(* IEC 61131-3 sources: SmartHomeNew/snapshots/2026-04-22, 17 files *)

(* ---- E_TwoFactor_Method.dut ---- *)
{attribute 'strict'}
TYPE E_TwoFactor_Method :
(
    TF_METHOD_NONE := 0,
    TF_METHOD_RFID := 1,
    TF_METHOD_TOTP := 2,
    TF_METHOD_BOTH := 3
) USINT;
END_TYPE

(* ---- ST_Heating_Config.dut ---- *)
{attribute 'pack_mode' := '1'}
TYPE ST_Heating_Config :
STRUCT
    Weather_Comp_Enabled : BOOL := TRUE;
    Weather_Coef : REAL := 0.1;
    Freeze_Threshold : REAL := 7.0;
    Overheat_Threshold : REAL := 45.0;
    Night_Reduction : REAL := 3.0;
    Target_Floor_Temp : REAL := 28.0;
    Target_Room_Temp : REAL := 22.0;
    Hysteresis : REAL := 0.5;
END_STRUCT
END_TYPE

(* ---- ST_System_State_Snapshot.dut ---- *)
{attribute 'pack_mode' := '1'}
TYPE ST_System_State_Snapshot :
STRUCT
    System_Time_MS : UDINT;
    Current_Scenario : E_SCENARIO_TYPE;
    Security_Armed : BOOL;
    Active_Alarms : INT;
    // Критические состояния для синхронизации
    Zone_Valves : ARRAY[1..8] OF BOOL;
    Manifold_Pumps : ARRAY[1..GVL_CONSTANTS.C_MAX_MANIFOLDS] OF BOOL;
    Lighting_States : ARRAY[1..32] OF BYTE;
    Blinds_Positions : ARRAY[1..GVL_CONSTANTS.C_MAX_BLINDS] OF BYTE;
    Socket_States : ARRAY[1..GVL_CONSTANTS.C_MAX_SOCKETS] OF BOOL;
    Gas_Valve_Closed : BOOL;
    Water_Valves_Closed : BOOL;
    Version : UDINT; // Версия состояния для разрешения конфликтов
END_STRUCT
END_TYPE

(* ---- ST_Zone_Sensors.dut ---- *)
{attribute 'pack_mode' := '1'}
TYPE ST_Zone_Sensors :
STRUCT
    Temp_Room : REAL;
    Temp_Floor : REAL;
    Motion_Active : BOOL;
    Switch_Physical : BOOL;
    Light_State : BOOL;
    Maintenance : ST_Component_Maintenance;
END_STRUCT
END_TYPE

(* ---- FB_Fault_Logger.st ---- *)
FUNCTION_BLOCK FB_Fault_Logger
VAR_INPUT
    VI_Severity  : E_System_Severity;
    VI_RootCause : E_System_Root_Cause;
    VI_Time_MS   : UDINT;
END_VAR

VAR_OUTPUT
    VO_Last_Event_Text : STRING(200);
    VO_Event_Count     : UINT;
    VO_Last_Index      : UINT;

    VO_Event_Time_MS   : ARRAY[1..16] OF UDINT;
    VO_Event_Severity  : ARRAY[1..16] OF E_System_Severity;
    VO_Event_RootCause : ARRAY[1..16] OF E_System_Root_Cause;
    VO_Event_Text      : ARRAY[1..16] OF STRING(200);
END_VAR

VAR
    L_Last_Severity  : E_System_Severity;
    L_Last_RootCause : E_System_Root_Cause;
    L_Write_Index    : UINT := 0;
    L_Event_Text     : STRING(200);
END_VAR

L_Event_Text := '';

IF (VI_Severity <> L_Last_Severity) OR (VI_RootCause <> L_Last_RootCause) THEN
    CASE VI_RootCause OF
        E_System_Root_Cause.ROOT_FIRE:
            L_Event_Text := 'EVENT: FIRE DETECTED';
        E_System_Root_Cause.ROOT_GAS_LEAK:
            L_Event_Text := 'EVENT: GAS LEAK';
        E_System_Root_Cause.ROOT_CO_CRITICAL:
            L_Event_Text := 'EVENT: CO CRITICAL';
        E_System_Root_Cause.ROOT_CO_WARNING:
            L_Event_Text := 'EVENT: CO WARNING';
        E_System_Root_Cause.ROOT_WATER_LEAK:
            L_Event_Text := 'EVENT: WATER LEAK';
        E_System_Root_Cause.ROOT_SENSOR_FAULT:
            L_Event_Text := 'EVENT: SENSOR FAULT';
        E_System_Root_Cause.ROOT_IO_OFFLINE:
            L_Event_Text := 'EVENT: IO OFFLINE';
        E_System_Root_Cause.ROOT_COMM_FAULT:
            L_Event_Text := 'EVENT: COMM FAULT';
        E_System_Root_Cause.ROOT_WATCHDOG_FAULT:
            L_Event_Text := 'EVENT: WATCHDOG FAULT';
        E_System_Root_Cause.ROOT_SUBSYSTEM_FAULT:
            L_Event_Text := 'EVENT: SUBSYSTEM FAULT';
        ELSE
            L_Event_Text := 'EVENT: SYSTEM STATE CHANGE';
    END_CASE;

    L_Write_Index := L_Write_Index + 1;
    IF L_Write_Index > 16 THEN
        L_Write_Index := 1;
    END_IF;

    VO_Event_Time_MS[L_Write_Index] := VI_Time_MS;
    VO_Event_Severity[L_Write_Index] := VI_Severity;
    VO_Event_RootCause[L_Write_Index] := VI_RootCause;
    VO_Event_Text[L_Write_Index] := L_Event_Text;

    VO_Last_Index := L_Write_Index;
    VO_Last_Event_Text := L_Event_Text;

    IF VO_Event_Count < 16 THEN
        VO_Event_Count := VO_Event_Count + 1;
    END_IF;
END_IF;

L_Last_Severity := VI_Severity;
L_Last_RootCause := VI_RootCause;
// >>> BULK_SYNC_ANCHOR: FB_Fault_Logger <<<

(* ---- FB_HMAC_SHA1.st ---- *)
FUNCTION_BLOCK FB_HMAC_SHA1
VAR_INPUT
    KeyLength : INT;
    MessageLength : INT;
END_VAR
VAR_IN_OUT
    Key : ARRAY[0..63] OF BYTE;
    Message : ARRAY[0..7] OF BYTE;
END_VAR
VAR_OUTPUT
    Hash : ARRAY[0..19] OF BYTE;
    Done : BOOL;
END_VAR
VAR
    i : INT;
    K_ipad : ARRAY[0..63] OF BYTE;
    K_opad : ARRAY[0..63] OF BYTE;
    InnerData : ARRAY[0..127] OF BYTE; // 64 (ipad) + 8 (msg)
    OuterData : ARRAY[0..127] OF BYTE; // 64 (opad) + 20 (inner hash)
    InnerHash : ARRAY[0..19] OF BYTE;
    FB_SHA1_Inner : FB_SHA1;
    FB_SHA1_Outer : FB_SHA1;
END_VAR

// 1. Prepare K_ipad and K_opad
FOR i := 0 TO 63 DO
    IF i < KeyLength THEN
        K_ipad[i] := Key[i] XOR 16#36;
        K_opad[i] := Key[i] XOR 16#5C;
    ELSE
        K_ipad[i] := 16#36;
        K_opad[i] := 16#5C;
    END_IF;
END_FOR;

// 2. Inner Hash: SHA1(K_ipad || Message)
FOR i := 0 TO 63 DO
    InnerData[i] := K_ipad[i];
END_FOR;
FOR i := 0 TO MessageLength - 1 DO
    InnerData[64 + i] := Message[i];
END_FOR;

FB_SHA1_Inner(Data := InnerData, Length := 64 + MessageLength, Hash => InnerHash);

// 3. Outer Hash: SHA1(K_opad || InnerHash)
FOR i := 0 TO 63 DO
    OuterData[i] := K_opad[i];
END_FOR;
FOR i := 0 TO 19 DO
    OuterData[64 + i] := InnerHash[i];
END_FOR;

FB_SHA1_Outer(Data := OuterData, Length := 84, Hash => Hash);

Done := TRUE;

(* ---- FB_NVRAM_Manager.st ---- *)
FUNCTION_BLOCK FB_NVRAM_Manager
VAR_INPUT
    VI_Command                  : BYTE; // 1=WRITE (READ not implemented)
    VI_Offset                   : UDINT; // Смещение в байтах
    VI_DataRef                  : REFERENCE TO BYTE;
    VI_DataSize                 : UDINT; // КРИТИЧНО: используем этот размер вместо SIZEOF
    VI_System_Time_MS           : UDINT;
    VI_Operator_ID              : STRING(10);
    VI_IsActivePLC              : BOOL;
    VI_TwoPersonConfirmation    : BOOL;
END_VAR
VAR_OUTPUT
    VO_Done                     : BOOL;
    VO_Error                    : BOOL;
    VO_ErrorID                  : UDINT;
    // VO_ReadDataRef removed (REFERENCE TO not allowed in output)
    VO_HMI_Status_Message       : STRING(200);
END_VAR
VAR
    L_prev_Command              : BYTE;
    L_cmd_rising                : BOOL;
    L_i                         : UDINT;
    L_Data_Changed              : BOOL; // Флаг изменения данных
    L_pData                      : POINTER TO BYTE;
END_VAR
VAR CONSTANT
    C_MAX_NVRAM_SIZE            : UDINT := 12800;
END_VAR

// Детекция фронта команды
L_cmd_rising := (VI_Command <> 0) AND (L_prev_Command = 0);
L_prev_Command := VI_Command;

IF L_cmd_rising THEN
    VO_Done := FALSE;
    VO_Error := FALSE;
    VO_ErrorID := 0;
    VO_HMI_Status_Message := '';

    // Валидация смещения
    IF VI_Offset >= C_MAX_NVRAM_SIZE THEN
        VO_Error := TRUE;
        VO_ErrorID := 16#1501;
        VO_HMI_Status_Message := 'NVRAM: Неверное смещение';
        VO_Done := TRUE;
        RETURN;
    END_IF;

    // Валидация указателя
    IF NOT __ISVALIDREF(VI_DataRef) THEN
        VO_Error := TRUE;
        VO_ErrorID := 16#150A;
        VO_HMI_Status_Message := 'NVRAM: Недействительная ссылка на данные';
        VO_Done := TRUE;
        RETURN;
    END_IF;

    L_pData := ADR(VI_DataRef);

    IF (VI_Offset + VI_DataSize) > C_MAX_NVRAM_SIZE THEN
        VO_Error := TRUE;
        VO_ErrorID := 16#150B;
        VO_HMI_Status_Message := 'NVRAM: Размер данных превышает доступный объем';
        VO_Done := TRUE;
        RETURN;
    END_IF;

    IF VI_Command = 2 THEN
    VO_Error := TRUE;
    VO_ErrorID := 16#150D;
    VO_HMI_Status_Message := 'NVRAM: READ not implemented';
    VO_Done := TRUE;
    RETURN;
END_IF;

IF VI_Command = 1 THEN // ЗАПИСЬ (WRITE)
        IF NOT VI_IsActivePLC THEN
            VO_Error := TRUE;
            VO_ErrorID := 16#1509;
            VO_HMI_Status_Message := 'NVRAM: Запись запрещена (STANDBY)';
        ELSE
            // Проверка на изменение данных перед записью
            L_Data_Changed := FALSE;
            FOR L_i := 0 TO VI_DataSize - 1 DO
                IF GVL_Retain.G_NVRAM_Data[VI_Offset + L_i] <> L_pData[L_i] THEN
                    L_Data_Changed := TRUE;
                    EXIT;
                END_IF;
            END_FOR;

            IF L_Data_Changed THEN
                // Безопасное копирование (WRITE)
                FOR L_i := 0 TO VI_DataSize - 1 DO
                    GVL_Retain.G_NVRAM_Data[VI_Offset + L_i] := L_pData[L_i];
                END_FOR;
                VO_HMI_Status_Message := 'NVRAM: Данные успешно сохранены в RETAIN';
            ELSE
                VO_HMI_Status_Message := 'NVRAM: Данные не изменились, запись пропущена';
            END_IF;
        END_IF;
        VO_Done := TRUE;
    END_IF;
END_IF;

IF VI_Command = 0 THEN
    VO_Done := FALSE;
END_IF;
// >>> BULK_SYNC_ANCHOR: FB_NVRAM_Manager <<<

(* ---- FB_Persist_Builder.st ---- *)
FUNCTION_BLOCK FB_Persist_Builder
VAR_IN_OUT
    VIO_PersistStruct : ST_Persist;
END_VAR

// === BUILD STRUCT FROM STATE ===
// === NVRAM SNAPSHOT VIA STRUCT ADAPTER ===
VIO_PersistStruct.System_Mode := GVL_STATE.G_System_Mode;

VIO_PersistStruct.Safety_Gas_Latched := GVL_STATE.G_Safety_Gas_Latched;
VIO_PersistStruct.Safety_Smoke_Latched := GVL_STATE.G_Safety_Smoke_Latched;
VIO_PersistStruct.Safety_Leak_Latched := GVL_STATE.G_Safety_Leak_Latched;

VIO_PersistStruct.DHW_Heating_Pump := GVL_STATE.G_DHW_Heating_Pump;
VIO_PersistStruct.Valid := TRUE;

// mirror to legacy persistent variables
GVL_PERSISTENT.P_System_Mode := VIO_PersistStruct.System_Mode;

GVL_PERSISTENT.P_Safety_Gas_Latched := VIO_PersistStruct.Safety_Gas_Latched;
GVL_PERSISTENT.P_Safety_Smoke_Latched := VIO_PersistStruct.Safety_Smoke_Latched;
GVL_PERSISTENT.P_Safety_Leak_Latched := VIO_PersistStruct.Safety_Leak_Latched;

GVL_PERSISTENT.P_DHW_Heating_Active := VIO_PersistStruct.DHW_Heating_Pump;
GVL_PERSISTENT.P_Valid := VIO_PersistStruct.Valid;

(* ---- FB_Persist_Pipeline.st ---- *)
FUNCTION_BLOCK FB_Persist_Pipeline
VAR_INPUT
    VI_PersistStruct : ST_Persist;
    VI_System_Time_MS : UDINT;
    VI_IsActivePLC : BOOL;
END_VAR
VAR_IN_OUT
    VIO_Apply_Settings : BOOL;
    VIO_Persist_Buffer : ARRAY[0..4] OF BYTE;
    VIO_Last_Written_Persist_Buffer : ARRAY[0..4] OF BYTE;
    VIO_Last_Persist_Write_MS : UDINT;
END_VAR
VAR_OUTPUT
    VO_NVRAM_Cmd : BYTE;
    VO_NVRAM_Offset : UDINT;
    VO_NVRAM_Done : BOOL;
    VO_NVRAM_Err : BOOL;
    VO_NVRAM_ErrID : UDINT;
END_VAR
VAR
    fbNVRAMManager : FB_NVRAM_Manager;
    L_Persist_Buffer_Changed : BOOL;
END_VAR

// === SERIALIZE PERSIST STRUCT → BUFFER ===

// System Mode
VIO_Persist_Buffer[0] := TO_BYTE(TO_INT(VI_PersistStruct.System_Mode));

// Gas
IF VI_PersistStruct.Safety_Gas_Latched THEN
    VIO_Persist_Buffer[1] := BYTE#1;
ELSE
    VIO_Persist_Buffer[1] := BYTE#0;
END_IF;

// Smoke
IF VI_PersistStruct.Safety_Smoke_Latched THEN
    VIO_Persist_Buffer[2] := BYTE#1;
ELSE
    VIO_Persist_Buffer[2] := BYTE#0;
END_IF;

// Leak
IF VI_PersistStruct.Safety_Leak_Latched THEN
    VIO_Persist_Buffer[3] := BYTE#1;
ELSE
    VIO_Persist_Buffer[3] := BYTE#0;
END_IF;

// DHW Pump
IF VI_PersistStruct.DHW_Heating_Pump THEN
    VIO_Persist_Buffer[4] := BYTE#1;
ELSE
    VIO_Persist_Buffer[4] := BYTE#0;
END_IF;

// === END SERIALIZE ===

L_Persist_Buffer_Changed :=
    (VIO_Persist_Buffer[0] <> VIO_Last_Written_Persist_Buffer[0]) OR
    (VIO_Persist_Buffer[1] <> VIO_Last_Written_Persist_Buffer[1]) OR
    (VIO_Persist_Buffer[2] <> VIO_Last_Written_Persist_Buffer[2]) OR
    (VIO_Persist_Buffer[3] <> VIO_Last_Written_Persist_Buffer[3]) OR
    (VIO_Persist_Buffer[4] <> VIO_Last_Written_Persist_Buffer[4]);

VO_NVRAM_Cmd := 0;
VO_NVRAM_Offset := 0;

IF VIO_Apply_Settings THEN
    // explicit config apply requests a controlled write
    // keep flag set until successful write confirmation
    VO_NVRAM_Cmd := 1;

ELSIF L_Persist_Buffer_Changed THEN
    // controlled write: no more often than once per 60 seconds
    IF (VIO_Last_Persist_Write_MS = 0) OR
       ((VI_System_Time_MS - VIO_Last_Persist_Write_MS) >= 60000) THEN
        VO_NVRAM_Cmd := 1;
    END_IF;
END_IF;

fbNVRAMManager(
    VI_Command := VO_NVRAM_Cmd,
    VI_Offset := VO_NVRAM_Offset,
    VI_DataRef := VIO_Persist_Buffer[0],
    VI_DataSize := 5,
    VI_System_Time_MS := VI_System_Time_MS,
    VI_Operator_ID := 'SYSTEM',
    VI_IsActivePLC := VI_IsActivePLC,
    VI_TwoPersonConfirmation := FALSE,
    VO_Done => VO_NVRAM_Done,
    VO_Error => VO_NVRAM_Err,
    VO_ErrorID => VO_NVRAM_ErrID
);

IF (VO_NVRAM_Cmd = 1) AND VO_NVRAM_Done AND NOT VO_NVRAM_Err THEN
    VIO_Last_Written_Persist_Buffer[0] := VIO_Persist_Buffer[0];
    VIO_Last_Written_Persist_Buffer[1] := VIO_Persist_Buffer[1];
    VIO_Last_Written_Persist_Buffer[2] := VIO_Persist_Buffer[2];
    VIO_Last_Written_Persist_Buffer[3] := VIO_Persist_Buffer[3];
    VIO_Last_Written_Persist_Buffer[4] := VIO_Persist_Buffer[4];
    VIO_Last_Persist_Write_MS := VI_System_Time_MS;
    VIO_Apply_Settings := FALSE;
END_IF;

(* ---- FB_Trend_Adapter.st ---- *)
FUNCTION_BLOCK FB_Trend_Adapter
VAR_INPUT
    VI_Data : ST_Trend_Data;
END_VAR

VAR_OUTPUT
    VO_Average : REAL;
    VO_Min : REAL;
    VO_Max : REAL;
    VO_Trend_Up : BOOL;
    VO_Trend_Down : BOOL;
END_VAR

VAR
    fbAnalyzer : FB_Trend_Analyzer;
    L_Data_Copy : ARRAY[1..GVL_CONSTANTS.C_MAX_TREND_DATA_POINTS] OF REAL;
    L_Count : INT;
    L_i : INT;
END_VAR

// Normalize count to analyzer bounds
L_Count := UDINT_TO_INT(VI_Data.record_count);
IF L_Count < 0 THEN
    L_Count := 0;
END_IF;
IF L_Count > GVL_CONSTANTS.C_MAX_TREND_DATA_POINTS THEN
    L_Count := GVL_CONSTANTS.C_MAX_TREND_DATA_POINTS;
END_IF;

// Copy source values into analyzer-compatible buffer
FOR L_i := 1 TO GVL_CONSTANTS.C_MAX_TREND_DATA_POINTS DO
    L_Data_Copy[L_i] := 0.0;
END_FOR;

IF L_Count > 0 THEN
    FOR L_i := 1 TO L_Count DO
        L_Data_Copy[L_i] := VI_Data.values[L_i];
    END_FOR;
END_IF;

fbAnalyzer(
    VI_Count := L_Count,
    VI_Data := L_Data_Copy,
    VO_Average => VO_Average,
    VO_Max => VO_Max,
    VO_Min => VO_Min,
    VO_Trend_Up => VO_Trend_Up,
    VO_Trend_Down => VO_Trend_Down
);

(* ---- FB_Trend_Analyzer.st ---- *)
FUNCTION_BLOCK FB_Trend_Analyzer
VAR_INPUT
    VI_Count      : INT;
END_VAR
VAR_IN_OUT
    VI_Data       : ARRAY[1..GVL_CONSTANTS.C_MAX_TREND_DATA_POINTS] OF REAL;
END_VAR
VAR_OUTPUT
    VO_Average    : REAL;
    VO_Max        : REAL;
    VO_Min        : REAL;
    VO_Trend_Up   : BOOL;
    VO_Trend_Down : BOOL;
END_VAR
VAR
    L_i   : INT;
    L_Sum : REAL;
END_VAR

IF VI_Count > 0 AND VI_Count <= GVL_CONSTANTS.C_MAX_TREND_DATA_POINTS THEN
    VO_Max := VI_Data[1];
    VO_Min := VI_Data[1];
    L_Sum := 0.0;

    FOR L_i := 1 TO VI_Count DO
        IF VI_Data[L_i] > VO_Max THEN VO_Max := VI_Data[L_i]; END_IF;
        IF VI_Data[L_i] < VO_Min THEN VO_Min := VI_Data[L_i]; END_IF;
        L_Sum := L_Sum + VI_Data[L_i];
    END_FOR;

    VO_Average := L_Sum / INT_TO_REAL(VI_Count);

    IF VI_Count >= 2 THEN
        VO_Trend_Up := (VI_Data[VI_Count] > VI_Data[1]);
        VO_Trend_Down := (VI_Data[VI_Count] < VI_Data[1]);
    END_IF;
END_IF;

(* ---- FB_Trend_Logger.st ---- *)
FUNCTION_BLOCK FB_Trend_Logger
VAR_INPUT
    VI_System_Time_MS : UDINT;
    VI_Config : ST_Trend_Config;
    VI_Current_Value : REAL;
END_VAR
VAR_OUTPUT
    VO_Data : ST_Trend_Data;
END_VAR
VAR
    L_Last_Log_Time : UDINT;
    L_Last_Value : REAL;
    L_Deviation : REAL;
END_VAR

IF NOT VI_Config.enabled THEN RETURN; END_IF;

// Логирование по изменению (Deadband) или по времени (раз в час)
L_Deviation := ABS(VI_Current_Value - L_Last_Value);
IF (L_Deviation >= (L_Last_Value * VI_Config.deviation_threshold_percent / 100.0)) OR
   ((SEL(VI_System_Time_MS >= L_Last_Log_Time, VI_System_Time_MS - L_Last_Log_Time, (4294967295 - L_Last_Log_Time) + VI_System_Time_MS + 1)) >= GVL_CONSTANTS.C_MS_IN_HOUR) THEN

    // Запись в массив
    VO_Data.write_index := (VO_Data.record_count MOD 100) + 1;
    VO_Data.values[VO_Data.write_index] := VI_Current_Value;
    VO_Data.timestamps[VO_Data.write_index] := VI_System_Time_MS;

    VO_Data.record_count := VO_Data.record_count + 1;
    VO_Data.sum_values := VO_Data.sum_values + VI_Current_Value;

    L_Last_Value := VI_Current_Value;
    L_Last_Log_Time := VI_System_Time_MS;
END_IF;

(* ---- FB_Ventilation_System_Manager.st ---- *)
FUNCTION_BLOCK FB_Ventilation_System_Manager
VAR_INPUT
    VI_System_Time_MS : UDINT; // Системное время (мс)
    VI_IsActivePLC : BOOL; // Флаг: Данный ПЛК является ведущим
    VI_Outdoor_Temp : REAL; // Уличная температура воздуха (°C)
    VI_Current_Scenario : E_SCENARIO_TYPE; // Текущий глобальный сценарий
    VI_System_Mode : E_System_Operating_Mode; // Агрегированный режим работы системы
    VI_Config : ST_Ventilation_Global_Config; // Конфигурация системы вентиляции
    VI_Fire_Alarm : BOOL; // Сигнал пожарной тревоги
    VI_Gas_Alarm : BOOL; // Сигнал газовой тревоги
    VI_PV3_Boost_Req : BOOL; // Запрос форсирования ПВ-3 от газоанализатора (ТЗ 5.1)
    VI_Supply_100_Req : BOOL; // Запрос 100% притока (ТЗ 6.4)
    VI_Exhaust_100_Req : BOOL; // Запрос 100% вытяжки (ТЗ 6.4)
    VI_Supply_80_Req : BOOL; // Запрос 80% притока (ТЗ 5.4)
    VI_Vent_Stop : BOOL; // Запрос на остановку вентиляции (ТЗ 5.3)
    VI_IO_Modules_Online : ARRAY[1..GVL_CONSTANTS.C_MAX_MODULES] OF BOOL; // Статусы модулей ввода-вывода (только чтение)
END_VAR
VAR_IN_OUT
    VI_Supply_Temps : ARRAY[1..GVL_CONSTANTS.C_MAX_SUPPLY_TEMPS] OF REAL; // Температура приточного воздуха после калорифера
    VI_Room_Temps : ARRAY[1..16] OF REAL; // Температура в помещениях (°C)
    VI_Room_Humidities : ARRAY[1..16] OF REAL; // Влажность в помещениях (%)
    VI_Room_CO2 : ARRAY[1..16] OF REAL; // Уровень CO2 в помещениях (ppm)
    VI_Wet_Zone_Active : ARRAY[1..GVL_CONSTANTS.C_MAX_WET_ZONES] OF BOOL; // Сигналы включения света в санузлах (ТЗ 4.0)
    VI_Rule_Actions : ARRAY[1..GVL_CONSTANTS.C_MAX_RULES] OF ST_Rule_Action; // Действия от Rule Engine
END_VAR
VAR_OUTPUT
    VO_Supply_Fans : ARRAY[1..GVL_CONSTANTS.C_MAX_SUPPLY_FANS] OF BYTE; // Выход: Управление приточными вентиляторами (0-100%)
    VO_Exhaust_Fans : ARRAY[1..GVL_CONSTANTS.C_MAX_EXHAUST_FANS] OF BYTE; // Выход: Управление вытяжными вентиляторами (0-100%)
    VO_Heater_Power : ARRAY[1..GVL_CONSTANTS.C_MAX_BOILERS] OF REAL; // Выход: Мощность калориферов (0-100%)
    VO_Status_Msg : STRING(200); // Строковое сообщение о статусе
END_VAR
VAR
    L_Policy_Normal : BOOL;
    L_Policy_Safe_Stop : BOOL;
    L_Policy_Degraded : BOOL;
    L_Policy_Freeze_Protection : BOOL;
    L_i : INT;
    L_j : INT;
    L_Max_CO2 : REAL;
    L_Max_Hum : REAL;
    L_Base_Speed : BYTE;
    L_Target_Temp : REAL;
    L_PID_Heaters : ARRAY[1..GVL_CONSTANTS.C_MAX_BOILERS] OF FB_PID_Controller;
    L_Wet_Zone_Timers : ARRAY[1..GVL_CONSTANTS.C_MAX_WET_ZONES] OF FB_System_Timer_TOF; // Таймеры выбега для вытяжек санузлов
END_VAR

// ========================================
// Ventilation policy layer
// ========================================
GVL_STATE.G_Ventilation_IO_Fault := FALSE;
GVL_STATE.G_Ventilation_Subsystem_Degraded := FALSE;
L_Policy_Normal := (VI_System_Mode = E_System_Operating_Mode.MODE_NORMAL);
L_Policy_Safe_Stop := (VI_System_Mode = E_System_Operating_Mode.MODE_SAFE_STOP);
L_Policy_Degraded := (VI_System_Mode = E_System_Operating_Mode.MODE_DEGRADED);
L_Policy_Freeze_Protection := (VI_System_Mode = E_System_Operating_Mode.MODE_FREEZE_PROTECTION);

IF NOT VI_IsActivePLC THEN
    FOR L_i := 1 TO GVL_CONSTANTS.C_MAX_SUPPLY_FANS DO
        VO_Supply_Fans[L_i] := 0;
        IF L_i <= GVL_CONSTANTS.C_MAX_SUPPLY_TEMPS THEN
            VO_Heater_Power[L_i] := 0.0;
        END_IF;
    END_FOR;
    FOR L_i := 1 TO GVL_CONSTANTS.C_MAX_EXHAUST_FANS DO
        VO_Exhaust_Fans[L_i] := 0;
    END_FOR;
    VO_Status_Msg := 'ВЕНТИЛЯЦИЯ: РЕЗЕРВНЫЙ ПЛК';
    RETURN;
END_IF;

// Проверка связи с модулями ввода-вывода
FOR L_i := 1 TO GVL_CONSTANTS.C_MAX_MODULES DO
    IF NOT VI_IO_Modules_Online[L_i] THEN
        GVL_STATE.G_Ventilation_IO_Fault := TRUE;
        // Переход в безопасное состояние при потере связи (отключение вентиляции)
        FOR L_j := 1 TO GVL_CONSTANTS.C_MAX_SUPPLY_FANS DO
            VO_Supply_Fans[L_j] := 0;
        END_FOR;
        FOR L_j := 1 TO GVL_CONSTANTS.C_MAX_EXHAUST_FANS DO
            VO_Exhaust_Fans[L_j] := 0;
        END_FOR;
        FOR L_j := 1 TO GVL_CONSTANTS.C_MAX_BOILERS DO
            VO_Heater_Power[L_j] := 0.0;
        END_FOR;
        VO_Status_Msg := 'ОШИБКА: Потеря связи с модулями ввода-вывода';
        RETURN;
    END_IF;
END_FOR;

// =========================
// SYSTEM MODE OVERRIDE
// =========================
// VENT_POLICY_ROUTING_PHASE3_V2
IF L_Policy_Safe_Stop THEN
    FOR L_i := 1 TO GVL_CONSTANTS.C_MAX_SUPPLY_FANS DO
        VO_Supply_Fans[L_i] := 0;
    END_FOR;
    FOR L_i := 1 TO GVL_CONSTANTS.C_MAX_EXHAUST_FANS DO
        VO_Exhaust_Fans[L_i] := 0;
    END_FOR;
    FOR L_i := 1 TO GVL_CONSTANTS.C_MAX_BOILERS DO
        VO_Heater_Power[L_i] := 0.0;
    END_FOR;
    VO_Status_Msg := 'ВЕНТИЛЯЦИЯ: ОСТАНОВЛЕНА POLICY SAFE_STOP';
    RETURN;
END_IF;

IF L_Policy_Degraded THEN
    FOR L_i := 1 TO GVL_CONSTANTS.C_MAX_SUPPLY_FANS DO
        VO_Supply_Fans[L_i] := 0;
    END_FOR;
    FOR L_i := 1 TO GVL_CONSTANTS.C_MAX_BOILERS DO
        VO_Heater_Power[L_i] := 0.0;
    END_FOR;
    GVL_STATE.G_Ventilation_Subsystem_Degraded := TRUE;
    VO_Status_Msg := 'ВЕНТИЛЯЦИЯ: DEGRADED POLICY';
END_IF;

IF L_Policy_Freeze_Protection THEN
    FOR L_i := 1 TO GVL_CONSTANTS.C_MAX_SUPPLY_FANS DO
        VO_Supply_Fans[L_i] := 0;
    END_FOR;
    FOR L_i := 1 TO GVL_CONSTANTS.C_MAX_EXHAUST_FANS DO
        VO_Exhaust_Fans[L_i] := 0;
    END_FOR;
    FOR L_i := 1 TO GVL_CONSTANTS.C_MAX_BOILERS DO
        VO_Heater_Power[L_i] := 0.0;
    END_FOR;
    VO_Status_Msg := 'ВЕНТИЛЯЦИЯ: FREEZE_PROTECTION POLICY (stop)';
    RETURN;
END_IF;

// MODE_FREEZE_PROTECTION пока оставляем на текущей штатной логике

// 1. Определение базовой скорости и целевой температуры по сценарию (ТЗ 7.1)
CASE VI_Current_Scenario OF
    E_SCENARIO_TYPE.SCENARIO_AWAY:
        L_Base_Speed := VI_Config.Scenario_Modes[3].Base_Fan_Speed;
        L_Target_Temp := VI_Config.Scenario_Modes[3].Target_Temp;
    E_SCENARIO_TYPE.SCENARIO_SLEEP:
        L_Base_Speed := VI_Config.Scenario_Modes[2].Base_Fan_Speed;
        L_Target_Temp := VI_Config.Scenario_Modes[2].Target_Temp;
    ELSE // PRESENCE, MORNING, EVENING
        L_Base_Speed := VI_Config.Scenario_Modes[1].Base_Fan_Speed;
        L_Target_Temp := VI_Config.Scenario_Modes[1].Target_Temp;
END_CASE;

// 2. Логика управления приточными установками (П-1, П-2, П-3)
FOR L_i := 1 TO GVL_CONSTANTS.C_MAX_SUPPLY_FANS DO
    // ПИД-регулирование мощности электрического калорифера
    IF L_i <= GVL_CONSTANTS.C_MAX_SUPPLY_TEMPS THEN
        L_PID_Heaters[L_i](
            VI_SetPoint := L_Target_Temp,
            VI_ProcessValue := VI_Supply_Temps[L_i], // Используем датчик температуры после калорифера
            VI_Kp := 4.0, VI_Tn := 120.0, VI_Tv := 0.0,
            VI_Y_Min := 0.0, VI_Y_Max := 100.0, VI_Cycle_Time_S := 1.0,
            VO_Output => VO_Heater_Power[L_i]
        );
    END_IF;

    // Определение скорости приточного вентилятора
    VO_Supply_Fans[L_i] := L_Base_Speed;

    // Обработка действий от Rule Engine
    FOR L_j := 1 TO GVL_CONSTANTS.C_MAX_RULES DO
        IF VI_Rule_Actions[L_j].Active AND VI_Rule_Actions[L_j].Target_ID = L_i THEN
            IF VI_Rule_Actions[L_j].Action_Type = E_Rule_Action_Type.ACTION_SET_VENTILATION THEN
                VO_Supply_Fans[L_i] := REAL_TO_BYTE(VI_Rule_Actions[L_j].Value);
            END_IF;
        END_IF;
    END_FOR;

    // Requests are operational requests and must not be reported as subsystem degradation.
END_FOR;

// 3. Логика управления вытяжными установками (В-1 .. В-5)
FOR L_i := 1 TO GVL_CONSTANTS.C_MAX_EXHAUST_FANS DO
    VO_Exhaust_Fans[L_i] := L_Base_Speed;

    // ТЗ 4.0: Логика вытяжки в санузлах
    FOR L_j := 1 TO GVL_CONSTANTS.C_MAX_WET_ZONES DO
        IF VI_Config.wet_zone_to_exhaust_map[L_j] = L_i THEN
            // Включение по свету, выключение с задержкой 5 минут (используем TOF)
            L_Wet_Zone_Timers[L_j](IN := VI_Wet_Zone_Active[L_j], PT := T#5m, VI_System_Time_MS := VI_System_Time_MS);
            IF VI_Wet_Zone_Active[L_j] THEN
                VO_Exhaust_Fans[L_i] := 80; // Повышенная скорость при присутствии
            ELSIF L_Wet_Zone_Timers[L_j].Q THEN
                VO_Exhaust_Fans[L_i] := 50; // Скорость выбега (пока таймер TOF активен)
            END_IF;
        END_IF;
    END_FOR;

    // Requests are operational requests and must not be reported as subsystem degradation.
END_FOR;

// ========================================
// VENT_FINAL_CLAMP
// ========================================
IF L_Policy_Degraded THEN
    FOR L_i := 1 TO GVL_CONSTANTS.C_MAX_EXHAUST_FANS DO
        VO_Exhaust_Fans[L_i] := MIN(VO_Exhaust_Fans[L_i], VI_Config.Degraded_Exhaust_Limit);
    END_FOR;
END_IF;

// 4. Формирование статусного сообщения
IF L_Policy_Safe_Stop THEN
    VO_Status_Msg := 'ВЕНТИЛЯЦИЯ: ОСТАНОВЛЕНА POLICY SAFE_STOP';
ELSIF L_Policy_Freeze_Protection THEN
    VO_Status_Msg := 'ВЕНТИЛЯЦИЯ: FREEZE_PROTECTION POLICY (stop)';
ELSIF L_Policy_Degraded THEN
    VO_Status_Msg := 'ВЕНТИЛЯЦИЯ: DEGRADED POLICY';
ELSE
    VO_Status_Msg := 'Вентиляция работает в штатном режиме';
END_IF;
// >>> BULK_SYNC_ANCHOR: FB_Ventilation_System_Manager <<<

(* ---- PRG_Heating.st ---- *)
PROGRAM PRG_Heating

VAR
    L_Last_Mode : INT := 0; // 0=normal,1=preheat,2=freeze
    L_Mode_Hold_Timer : FB_System_Timer;
END_VAR

VAR
    fbHeatingManager : FB_Heating_System_Manager;
    fbDHWManager : FB_DHW_Manager;
    L_i : INT;
    L_Zone_Valves_8 : ARRAY[1..8] OF BOOL;
    L_Boiler_Modulation_REAL : ARRAY[1..GVL_CONSTANTS.C_MAX_BOILERS] OF REAL;
    L_Heating_Emergency_Stop : BOOL;
    L_Heating_Gas_Safety_Stop : BOOL;
    L_Heating_DHW_Demand : BOOL;
END_VAR

FOR L_i := 1 TO GVL_CONSTANTS.C_MAX_BOILERS DO
    L_Boiler_Modulation_REAL[L_i] := TO_REAL(GVL_IO.AI_Boiler_Modulation[L_i]);
END_FOR;

// === Heating Arbitration ===
L_Heating_Emergency_Stop := GVL_STATE.G_Safety_Emergency_Stop;
L_Heating_Gas_Safety_Stop := GVL_STATE.G_Safety_Gas_Latched;
L_Heating_DHW_Demand := fbDHWManager.VO_Heating_Pump;

// Priority 1: emergency stop
IF L_Heating_Emergency_Stop THEN
    L_Heating_Gas_Safety_Stop := FALSE;
    L_Heating_DHW_Demand := FALSE;
// Priority 2: gas safety stop
ELSIF L_Heating_Gas_Safety_Stop THEN
    L_Heating_DHW_Demand := FALSE;
ELSIF GVL_STATE.G_System_Mode = E_System_Operating_Mode.MODE_DEGRADED THEN
    L_Heating_DHW_Demand := FALSE;
END_IF;

// --- CONSOLIDATED HEATING REQUEST / ARBITRATION / STABILIZATION ---
L_Mode_Hold_Timer(
    IN := TRUE,
    PT := T#30s,
    VI_System_Time_MS := GVL_STATUS.G_System_Time_MS
);

IF L_Mode_Hold_Timer.Q THEN
    IF GVL_STATE.G_Freeze_Request THEN
        L_Last_Mode := 2; // freeze
    ELSIF GVL_STATE.G_Preheat_Request THEN
        L_Last_Mode := 1; // preheat
    ELSE
        L_Last_Mode := 0; // normal
    END_IF;
END_IF;

CASE L_Last_Mode OF
    2:
        GVL_STATE.G_Target_Temperature := 5.0;
    1:
        GVL_STATE.G_Target_Temperature := 22.0;
    ELSE
        GVL_STATE.G_Target_Temperature := 20.0;
END_CASE;

// 9. Управление климатом (Отопление)
fbHeatingManager(
    VI_Preheat_Request := GVL_HEATING_REQUEST.G_Preheat_Request,
    VI_System_Time_MS := GVL_STATUS.G_System_Time_MS,
    VI_Current_TOD := GVL_STATUS.G_Current_TOD,
    VI_IsActivePLC := GVL_STATUS.G_Is_Active_PLC,
    VI_Outdoor_Temp := GVL_STATE.G_Outdoor_Temp,
    VI_Floor_Temps := GVL_STATE.G_Floor_Temps,
    VI_Room_Temps := GVL_STATE.G_Room_Temps,
    VI_Config := GVL_CONFIG.G_Heating_Config,
    VI_Zone_Configs := GVL_CONFIG.G_HMI_FloorHeating_Configs,
    VI_Tariff := GVL_CONFIG.G_HMI_Tariff_Settings,
    VI_Current_Hour := TO_UINT(GVL_STATUS.G_Time_Of_Day_MS / GVL_CONSTANTS.C_MS_IN_HOUR),
    VI_Manifold_Pressures := GVL_STATE.G_Manifold_Pressures,
    VI_Manifold_Currents := GVL_STATE.G_Manifold_Currents,
    VI_Manifold_Temps_Supply := GVL_STATE.G_Manifold_T_Supply,
    VI_Manifold_Temps_Return := GVL_STATE.G_Manifold_T_Return,
    VI_Boiler_Flame_Status := GVL_STATE.G_Boiler_Flame,
    VI_Boiler_Error_Status := GVL_STATE.G_Boiler_Error,
    VI_Boiler_OT_Online := GVL_STATE.G_Boiler_OT_Online,
    VI_Boiler_Modulation := L_Boiler_Modulation_REAL,
    VI_Rule_Actions := GVL_STATE.G_Rule_Actions,
    VI_Boiler_Stop := FALSE, // legacy input disabled; safety flows via mode/latches
    VI_IO_Modules_Online := GVL_STATUS.G_IO_Modules_Online,
    VI_DHW_Heating_Demand := L_Heating_DHW_Demand,
    VI_DHW_Target_Temp := GVL_CONFIG.G_DHW_Config.Target_Temp,
    VI_Current_Scenario := GVL_STATUS.G_Current_Scenario,
    VI_System_Mode := GVL_STATE.G_System_Mode,
    VI_Emergency_Stop := L_Heating_Emergency_Stop,
    VI_Gas_Safety_Stop := L_Heating_Gas_Safety_Stop,
    VI_Scenario_Configs := GVL_CONFIG.G_HMI_Scenario_Configs,
    VI_Manifold_End_Switches := GVL_STATE.G_Manifold_End_Switches,
    VI_Valve_Test_Config := GVL_CONFIG.G_Valve_Test_Config,
    VO_Manifold_Valves => GVL_STATE.G_Manifold_Valves,
    VO_Manifold_Pumps => GVL_STATE.G_Manifold_Pumps,
    VO_Zone_Valves => L_Zone_Valves_8,
    VO_Boiler_OT_Enable => GVL_STATE.G_Boiler_OT_Enable,
    VO_Boiler_OT_Setpoint => GVL_STATE.G_Boiler_OT_Setpoint,
    VO_Backup_Circulation_Pump => GVL_STATE.G_Backup_Circulation_Pump,
    VO_Electric_Heater_Enable => GVL_STATE.G_Electric_Heater_Enable,
    VO_Freeze_Risk_Status => GVL_STATE.G_Safety_Freeze_Risk,
    VO_Status => GVL_STATUS.G_Manifold_Status,
    VO_Boiler_Status => GVL_STATUS.G_Boiler_Status
);

// 12. Управление ГВС
fbDHWManager(
    VI_System_Time_MS := GVL_STATUS.G_System_Time_MS,
    VI_Current_TOD := GVL_STATUS.G_Current_TOD,
    VI_IsActivePLC := GVL_STATUS.G_Is_Active_PLC,
    VI_Temp := GVL_STATE.G_DHW_Temp,
    VI_Pressure := GVL_STATE.G_DHW_Pressure,
    VI_Config := GVL_CONFIG.G_DHW_Config,
    VI_Current_Day_Of_Week := GVL_STATUS.G_Current_Day,
    VI_IO_Modules_Online := GVL_STATUS.G_IO_Modules_Online,
    VI_Reset_Errors := GVL_INTENT_USER.I_Reset_Errors,
    VI_Emergency_Stop := GVL_STATE.G_Safety_Emergency_Stop,
    VI_System_Mode := GVL_STATE.G_System_Mode,
    VO_Heating_Pump => GVL_STATE.G_DHW_Heating_Pump,
    VO_Circ_Pump => GVL_STATE.G_DHW_Circ_Pump,
    VO_Status => GVL_STATUS.G_DHW_Status
);

// Integrated freeze-hardware diagnostics and maintenance gating
GVL_STATUS.G_Diagnostics.Backup_Pump_Out_Of_Service := NOT GVL_CONFIG.G_Backup_Circulation_Pump_In_Service;
GVL_STATUS.G_Diagnostics.Electric_Heater_Out_Of_Service := NOT GVL_CONFIG.G_Electric_Heater_In_Service;
IF NOT GVL_CONFIG.G_Backup_Circulation_Pump_In_Service THEN
    GVL_STATE.G_Backup_Circulation_Pump := FALSE;
END_IF;
IF NOT GVL_CONFIG.G_Electric_Heater_In_Service THEN
    GVL_STATE.G_Electric_Heater_Enable := FALSE;
END_IF;

GVL_STATE.G_Freeze_Hardware_Degraded := GVL_STATUS.G_Diagnostics.Backup_Pump_Fault OR GVL_STATUS.G_Diagnostics.Electric_Heater_Fault;
GVL_STATE.G_Freeze_Hardware_Failed := GVL_STATUS.G_Diagnostics.Backup_Pump_Fault AND GVL_STATUS.G_Diagnostics.Electric_Heater_Fault;

IF GVL_STATE.G_Freeze_Hardware_Failed THEN
    GVL_STATE.G_Backup_Circulation_Pump := FALSE;
    GVL_STATE.G_Electric_Heater_Enable := FALSE;
    GVL_STATE.G_Safety_Freeze_Risk := TRUE;
END_IF;

FOR L_i := 1 TO GVL_CONSTANTS.C_MAX_MANIFOLDS DO
    GVL_STATUS.G_Diagnostics.Manifold_Pump_Out_Of_Service[L_i] := NOT GVL_CONFIG.G_Manifold_Pump_In_Service[L_i];
    IF NOT GVL_CONFIG.G_Manifold_Pump_In_Service[L_i] THEN
        GVL_STATE.G_Manifold_Pumps[L_i] := FALSE;
    END_IF;
END_FOR;
GVL_STATUS.G_Diagnostics.DHW_Heating_Pump_Out_Of_Service := NOT GVL_CONFIG.G_DHW_Heating_Pump_In_Service;
IF NOT GVL_CONFIG.G_DHW_Heating_Pump_In_Service THEN
    GVL_STATE.G_DHW_Heating_Pump := FALSE;
END_IF;
GVL_STATUS.G_Diagnostics.DHW_Circ_Pump_Out_Of_Service := NOT GVL_CONFIG.G_DHW_Circ_Pump_In_Service;
IF NOT GVL_CONFIG.G_DHW_Circ_Pump_In_Service THEN
    GVL_STATE.G_DHW_Circ_Pump := FALSE;
END_IF;
// >>> BULK_SYNC_ANCHOR: PRG_Heating <<<

// HEATING ADAPTER COPY OUT
FOR L_i := 1 TO 8 DO
    GVL_STATE.G_Zone_Valves[L_i] := L_Zone_Valves_8[L_i];
END_FOR;

(* ---- PRG_IO_Read.st ---- *)
PROGRAM PRG_IO_Read
VAR
    L_i : INT;
    L_Debounce_Time : TIME := T#100MS;

    fbDebounce_Switches : ARRAY[1..8] OF FB_System_Timer;
    fbDebounce_Motion : ARRAY[1..8] OF FB_System_Timer;
    fbDebounce_Security_Open : ARRAY[1..GVL_CONSTANTS.C_MAX_SECURITY_SENSORS] OF FB_System_Timer;
    fbDebounce_Security_Glass : ARRAY[1..GVL_CONSTANTS.C_MAX_SECURITY_SENSORS] OF FB_System_Timer;
    fbDebounce_Flood : ARRAY[1..GVL_CONSTANTS.C_MAX_FLOOD_SENSORS] OF FB_System_Timer;
    fbDebounce_Smoke : ARRAY[1..GVL_CONSTANTS.C_MAX_SMOKE_SENSORS] OF FB_System_Timer;
    fbDebounce_Group_2F : FB_System_Timer;

    fbIO_Watchdog_1 : FB_IO_Module_Watchdog;
    fbIO_Watchdog_2 : FB_IO_Module_Watchdog;
    L_IO_Error_Active : BOOL;
END_VAR

// 0. КОНТРОЛЬ СВЯЗИ С МОДУЛЯМИ ВВОДА-ВЫВОДА (Watchdog)
fbIO_Watchdog_1(
    VI_System_Time_MS := GVL_STATUS.G_System_Time_MS,
    VI_Module_ID := 1,
    VI_Heartbeat_Signal := GVL_IO.DI_Module_1_Heartbeat,
    VI_Timeout_MS := 2000
);

fbIO_Watchdog_2(
    VI_System_Time_MS := GVL_STATUS.G_System_Time_MS,
    VI_Module_ID := 2,
    VI_Heartbeat_Signal := GVL_IO.DI_Module_2_Heartbeat,
    VI_Timeout_MS := 2000
);

GVL_STATUS.G_IO_Modules_Online[1] := fbIO_Watchdog_1.VO_Module_Online;
GVL_STATUS.G_IO_Modules_Online[2] := fbIO_Watchdog_2.VO_Module_Online;

L_IO_Error_Active := fbIO_Watchdog_1.VO_Error_Active OR fbIO_Watchdog_2.VO_Error_Active;

IF L_IO_Error_Active THEN
    GVL_COMMAND.G_Gas_Valve_Close := TRUE;
    GVL_COMMAND.G_Close_Valve_35 := TRUE;
    GVL_COMMAND.G_Close_Valve_36 := TRUE;
    FOR L_i := 1 TO GVL_CONSTANTS.C_MAX_MANIFOLDS DO GVL_STATE.G_Manifold_Pumps[L_i] := FALSE; END_FOR;
END_IF;

// 1. ЧТЕНИЕ И ФИЛЬТРАЦИЯ ВХОДОВ
FOR L_i := 1 TO 8 DO
    fbDebounce_Switches[L_i](IN := GVL_IO.DI_Lighting_Switches[L_i], PT := L_Debounce_Time, VI_System_Time_MS := GVL_STATUS.G_System_Time_MS);
    GVL_STATE.G_Physical_Switches[L_i] := fbDebounce_Switches[L_i].Q;

    fbDebounce_Motion[L_i](IN := GVL_IO.DI_Motion_Sensors[L_i], PT := L_Debounce_Time, VI_System_Time_MS := GVL_STATUS.G_System_Time_MS);
    GVL_STATE.G_Motion_Sensors[L_i] := fbDebounce_Motion[L_i].Q;
END_FOR;

FOR L_i := 1 TO GVL_CONSTANTS.C_MAX_SOCKETS DO
    // В текущей концепции локальные физические выключатели розеток не используются.
    // Состояние оставляем FALSE для обратной совместимости структуры.
    GVL_STATE.G_Socket_Switches[L_i] := FALSE;
END_FOR;

FOR L_i := 1 TO GVL_CONSTANTS.C_MAX_SECURITY_SENSORS DO
    fbDebounce_Security_Open[L_i](IN := GVL_IO.DI_Security_Open[L_i], PT := L_Debounce_Time, VI_System_Time_MS := GVL_STATUS.G_System_Time_MS);
    fbDebounce_Security_Glass[L_i](IN := GVL_IO.DI_Security_Glass[L_i], PT := L_Debounce_Time, VI_System_Time_MS := GVL_STATUS.G_System_Time_MS);
END_FOR;
fbDebounce_Group_2F(IN := GVL_IO.DI_Security_2F_Group, PT := L_Debounce_Time, VI_System_Time_MS := GVL_STATUS.G_System_Time_MS);

FOR L_i := 1 TO GVL_CONSTANTS.C_MAX_DOOR_SENSORS DO
    IF GVL_CONFIG.G_Door_Map[L_i] > 0 AND GVL_CONFIG.G_Door_Map[L_i] <= GVL_CONSTANTS.C_MAX_SECURITY_SENSORS THEN
        GVL_STATE.G_Door_Sensors[L_i] := fbDebounce_Security_Open[GVL_CONFIG.G_Door_Map[L_i]].Q;
    END_IF;
END_FOR;

FOR L_i := 1 TO 8 DO
    IF GVL_CONFIG.G_Window_Map[L_i] > 0 THEN
        IF GVL_CONFIG.G_Window_Map[L_i] <= GVL_CONSTANTS.C_MAX_SECURITY_SENSORS THEN
            GVL_STATE.G_Window_Sensors[L_i] := fbDebounce_Security_Open[GVL_CONFIG.G_Window_Map[L_i]].Q;
        ELSIF GVL_CONFIG.G_Window_Map[L_i] <= (GVL_CONSTANTS.C_MAX_SECURITY_SENSORS * 2) THEN
            GVL_STATE.G_Window_Sensors[L_i] := fbDebounce_Security_Glass[GVL_CONFIG.G_Window_Map[L_i] - GVL_CONSTANTS.C_MAX_SECURITY_SENSORS].Q;
        END_IF;
    END_IF;
END_FOR;
GVL_STATE.G_Window_Sensors[16] := fbDebounce_Group_2F.Q;

FOR L_i := 1 TO GVL_CONSTANTS.C_MAX_FLOOD_SENSORS DO
    fbDebounce_Flood[L_i](IN := GVL_IO.DI_Flood_Sensors[L_i], PT := L_Debounce_Time, VI_System_Time_MS := GVL_STATUS.G_System_Time_MS);
    GVL_STATE.G_Water_Sensors[L_i] := fbDebounce_Flood[L_i].Q;
END_FOR;

FOR L_i := 1 TO GVL_CONSTANTS.C_MAX_SMOKE_SENSORS DO
    fbDebounce_Smoke[L_i](IN := GVL_IO.DI_Smoke_Sensors[L_i], PT := L_Debounce_Time, VI_System_Time_MS := GVL_STATUS.G_System_Time_MS);
    GVL_STATE.G_Smoke_Sensors[L_i] := fbDebounce_Smoke[L_i].Q;
END_FOR;

IF GVL_IO.AI_Temp_Outdoor.wStatus = 0 THEN
    GVL_STATE.G_Outdoor_Temp := GVL_IO.AI_Temp_Outdoor.rValue;
END_IF;

FOR L_i := 1 TO GVL_CONSTANTS.C_MAX_SUPPLY_TEMPS DO
    IF GVL_IO.AI_Supply_Temps[L_i].wStatus = 0 THEN
        GVL_STATE.G_Supply_Temps[L_i] := GVL_IO.AI_Supply_Temps[L_i].rValue;
    END_IF;
END_FOR;

FOR L_i := 1 TO 8 DO
    GVL_STATE.G_Room_Hum[L_i] := GVL_IO.AI_Room_Hum[L_i];
    GVL_STATE.G_Room_CO2[L_i] := GVL_IO.AI_Room_CO2[L_i];
END_FOR;
FOR L_i := 1 TO 8 DO
    IF GVL_CONFIG.G_FloorTemp_Map[L_i] > 0 AND GVL_CONFIG.G_FloorTemp_Map[L_i] <= 8 THEN
        GVL_STATE.G_Floor_Temps[L_i] := GVL_IO.AI_Floor_Temps[GVL_CONFIG.G_FloorTemp_Map[L_i]];
    END_IF;
    IF GVL_CONFIG.G_RoomTemp_Map[L_i] > 0 AND GVL_CONFIG.G_RoomTemp_Map[L_i] <= 8 THEN
        GVL_STATE.G_Room_Temps[L_i] := GVL_IO.AI_Room_Temps[GVL_CONFIG.G_RoomTemp_Map[L_i]];
    END_IF;
END_FOR;

FOR L_i := 1 TO GVL_CONSTANTS.C_MAX_MANIFOLDS DO
    GVL_STATE.G_Manifold_Pressures[L_i] := INT_TO_REAL(GVL_IO.AI_Manifold_Pressures[L_i]) / 10.0;
    GVL_STATE.G_Manifold_Currents[L_i] := INT_TO_REAL(GVL_IO.AI_Manifold_Currents[L_i]) / 100.0;
    IF GVL_IO.AI_Manifold_Temps_Supply[L_i].wStatus = 0 THEN
        GVL_STATE.G_Manifold_T_Supply[L_i] := GVL_IO.AI_Manifold_Temps_Supply[L_i].rValue;
    END_IF;
    GVL_STATE.G_Manifold_T_Return[L_i] := INT_TO_REAL(GVL_IO.AI_Manifold_Temps_Return[L_i]) / 10.0;
    GVL_STATE.G_Manifold_End_Switches[L_i] := GVL_IO.DI_Manifold_End_Switches[L_i];
END_FOR;

FOR L_i := 1 TO GVL_CONSTANTS.C_MAX_METHANE_SENSORS DO
    IF GVL_IO.AI_Methane_LEL[L_i].wStatus = 0 THEN
        GVL_STATE.G_Methane_Sensors[L_i] := GVL_IO.AI_Methane_LEL[L_i].rValue;
    END_IF;
END_FOR;
GVL_STATE.G_Boiler_Flame := GVL_IO.AI_Boiler_Flame_Status;
GVL_STATE.G_Boiler_Error := GVL_IO.DI_Boiler_Error;
// --- SAFETY bootstrap mapping (temporary, will be normalized later if dedicated managers exist) ---
GVL_STATE.G_Safety_Gas_Alarm := FALSE;
GVL_STATE.G_Safety_Leak_Alarm := FALSE;
GVL_STATE.G_Safety_Smoke_Alarm := FALSE;

// Временное безопасное поведение:
// до подключения реального драйвера/шлюза OpenTherm считаем канал котла недоступным.
FOR L_i := 1 TO GVL_CONSTANTS.C_MAX_BOILERS DO
    GVL_STATE.G_Boiler_OT_Online[L_i] := FALSE;
END_FOR;
GVL_STATE.G_CO_Sensors := GVL_IO.AI_CO_PPM;

GVL_STATE.G_DHW_Temp := GVL_IO.AI_DHW_Temp;
GVL_STATE.G_DHW_Pressure := GVL_IO.AI_DHW_Pressure;

// Water zonal valve feedback mapping
GVL_STATE.G_Water_Zone_Open_FB := GVL_IO.DI_Water_Zone_Open_FB;
GVL_STATE.G_Water_Zone_Close_FB := GVL_IO.DI_Water_Zone_Close_FB;

GVL_STATUS.G_Diagnostics.Backup_Pump_Fault := FALSE;
GVL_STATUS.G_Diagnostics.Electric_Heater_Fault := FALSE;
// >>> BULK_SYNC_ANCHOR: PRG_IO_Read <<<

(* ---- PRG_Lighting.st ---- *)
PROGRAM PRG_Lighting
VAR
    L_i : INT;
    fbLightingManager : FB_Lighting_Blinds_Manager;
    fbSocketManager : FB_Socket_Manager;
    L_Manual_Light_Override_32 : ARRAY[1..32] OF BYTE;
    L_Manual_Blinds_Override_32 : ARRAY[1..32] OF BYTE;
    L_Manual_Socket_Override_32 : ARRAY[1..32] OF BOOL;
    L_Sim_Lights_32 : ARRAY[1..32] OF BOOL;
    L_Physical_Switches_32 : ARRAY[1..32] OF BOOL;
    L_Motion_Sensors_32 : ARRAY[1..32] OF BOOL;

    // ADAPTER ARRAYS (match FB expected sizes)
    L_Blinds_Override : ARRAY[1..GVL_CONSTANTS.C_MAX_BLINDS] OF BYTE;
    L_Socket_Override : ARRAY[1..GVL_CONSTANTS.C_MAX_SOCKETS] OF BOOL;
END_VAR

FOR L_i := 1 TO 32 DO
    IF L_i <= 16 THEN
        IF GVL_INTENT_SYSTEM.I_Lighting_Overrides_Block THEN
            L_Manual_Light_Override_32[L_i] := 0;
        ELSE
            L_Manual_Light_Override_32[L_i] := GVL_INTENT_USER.I_Lighting_Override_32[L_i];
        END_IF;
        L_Sim_Lights_32[L_i] := GVL_STATE.G_Sim_Lights[L_i];
        L_Physical_Switches_32[L_i] := GVL_STATE.G_Physical_Switches[L_i];
        L_Motion_Sensors_32[L_i] := GVL_STATE.G_Motion_Sensors[L_i];
    ELSE
        L_Manual_Light_Override_32[L_i] := 0;
        L_Sim_Lights_32[L_i] := FALSE;
        L_Physical_Switches_32[L_i] := FALSE;
        L_Motion_Sensors_32[L_i] := FALSE;
    END_IF;

    IF GVL_INTENT_SYSTEM.I_Blinds_Overrides_Block THEN
        L_Manual_Blinds_Override_32[L_i] := 0;
    ELSE
        L_Manual_Blinds_Override_32[L_i] := GVL_INTENT_USER.I_Blinds_Override_32[L_i];
    END_IF;

    IF GVL_INTENT_SYSTEM.I_Socket_Overrides_Block THEN
        L_Manual_Socket_Override_32[L_i] := FALSE;
    ELSE
        L_Manual_Socket_Override_32[L_i] := GVL_INTENT_USER.I_Socket_Override_32[L_i];
    END_IF;
END_FOR;

// ADAPTER: copy to FB-sized arrays
FOR L_i := 1 TO GVL_CONSTANTS.C_MAX_BLINDS DO
    L_Blinds_Override[L_i] := L_Manual_Blinds_Override_32[L_i];
END_FOR;

FOR L_i := 1 TO GVL_CONSTANTS.C_MAX_SOCKETS DO
    L_Socket_Override[L_i] := L_Manual_Socket_Override_32[L_i];
END_FOR;

// 10. Управление освещением и шторами
fbLightingManager(
    VI_System_Time_MS := GVL_STATUS.G_System_Time_MS,
    VI_IsActivePLC := GVL_STATUS.G_Is_Active_PLC,
    VI_Current_Scenario := GVL_STATUS.G_Current_Scenario,
    VI_Away_Level := 1,
    VI_Simulation_Active := GVL_STATUS.G_Sim_Active,
    VI_Manual_Light_Override := L_Manual_Light_Override_32,
    VI_Manual_Blinds_Override := L_Blinds_Override,
    VI_Simulation_Lights := L_Sim_Lights_32,
    VI_Physical_Switches := L_Physical_Switches_32,
    VI_Motion_Sensors := L_Motion_Sensors_32,
    VI_Is_Night := GVL_STATUS.G_Is_Night,
    VI_Rule_Actions := GVL_STATE.G_Rule_Actions,
    VI_IO_Modules_Online := GVL_STATUS.G_IO_Modules_Online,
    VI_Wet_Zone_Map := GVL_CONFIG.G_Wet_Zone_Map,
    VI_Scenario_Configs := GVL_CONFIG.G_HMI_Scenario_Configs,
    VO_Lighting_Levels => GVL_STATE.G_Lighting_Levels,
    VO_Blinds_Positions => GVL_STATE.G_Blinds_Positions
);

// 11.5 Управление розетками
fbSocketManager(
    VI_System_Time_MS := GVL_STATUS.G_System_Time_MS,
    VI_IsActivePLC := GVL_STATUS.G_Is_Active_PLC,
    VI_Scenario := GVL_STATUS.G_Current_Scenario,
    VI_Manual_Override := L_Socket_Override,
    VI_Physical_Switches := GVL_STATE.G_Socket_Switches,
    VI_Rule_Actions := GVL_STATE.G_Rule_Actions,
    VI_Fire_Alarm := GVL_ALARM.G_Fire_Alarm_Active,
    VI_Flood_Alarm := GVL_ALARM.G_Flood_Alarm_Active,
    VI_Security_Armed := GVL_ALARM.G_Security_Armed,
    VI_IO_Modules_Online := GVL_STATUS.G_IO_Modules_Online,
    VO_Socket_States => GVL_STATE.G_Socket_States
);

// Evacuation lighting override
IF GVL_STATE.G_Evacuation_Lighting_Active THEN
    FOR L_i := 1 TO 8 DO
        IF (L_i MOD 2) = 0 THEN
            GVL_STATE.G_Lighting_Levels[L_i] := 100;
        ELSE
            GVL_STATE.G_Lighting_Levels[L_i] := 0;
        END_IF;
    END_FOR;
END_IF;

// Directional evacuation override
IF GVL_STATE.G_Evacuation_Lighting_Active THEN
    FOR L_i := 1 TO GVL_CONFIG.C_MAX_LIGHT_ZONES DO
        CASE GVL_STATE.G_Evac_Guidance[L_i] OF
            -1:
                GVL_STATE.G_Lighting_Levels[L_i] := 0;
            1:
                GVL_STATE.G_Lighting_Levels[L_i] := 100;
        ELSE
            GVL_STATE.G_Lighting_Levels[L_i] := SEL((L_i MOD 2) = 0, 0, 100);
        END_CASE;
    END_FOR;
END_IF;
// >>> BULK_SYNC_ANCHOR: PRG_Lighting <<<

(* ---- PRG_System.st ---- *)
PROGRAM PRG_System
VAR
    L_i : INT;
    L_Motion_Sensors_16 : ARRAY[1..16] OF BOOL;
    // --- ADAPTER LAYER ---
    L_Zone_Valves_8 : ARRAY[1..8] OF BOOL;
    L_Lighting_32   : ARRAY[1..32] OF BYTE;
    L_Lighting_Bool_32 : ARRAY[1..32] OF BOOL;
    L_FloorTemps_8  : ARRAY[1..8] OF REAL;
    fbCoreKernelObserver : FB_CoreKernel_Live_Observer;
    fbSystemHealth : FB_System_Health;
    fbRedundancy : FB_Redundancy_Manager;
    fbGateway : FB_Gateway_Interface;
    fbScenarioManager : FB_Scenario_Manager;
    fbSimulationManager : FB_Simulation_Manager;
    fbRuleEngine : FB_Rule_Engine;
    fbNVRAMManager : FB_NVRAM_Manager;

    fbBlackBox : FB_BlackBox_Recorder;
    fbAstroTimer : FB_Astro_Timer;
    fbAlarmManager : FB_Alarm_Manager;
    fbHistoryManager : FB_History_Manager;
    fbSafety : FB_Safety_Manager;
    fbStateManager : FB_State_Manager;
    fbWatchdog : FB_Watchdog;
    fbHMIInterface : FB_HMI_Interface;
    fbFaultLogger : FB_Fault_Logger;
    fbLogEvent : FB_LogEvent;

    L_Time_Diff : UDINT;
    L_Local_State : ST_System_State_Snapshot;
    L_Remote_State : ST_System_State_Snapshot;
    L_NVRAM_Cmd : BYTE;
    L_NVRAM_Offset : UDINT;
    L_NVRAM_Done : BOOL;
    L_NVRAM_Err : BOOL;
    L_NVRAM_ErrID : UDINT;
    L_BB_Record : ST_BlackBox_Record;
    L_BB_Freeze : BOOL;
    L_Scenario_Idx : INT;
        L_Last_Operator_Blocked : BOOL;
    L_Last_DHW_Heating_In_Service : BOOL;
    L_Last_DHW_Circ_In_Service : BOOL;
    L_Dangerous_Action_Armed : BOOL;
    L_Dangerous_Action_Deadline_MS : UDINT;
    L_Maintenance_Apply_Intent : BOOL;
    L_Last_System_Mode : E_System_Operating_Mode;
    L_Last_First_Fault_Type : INT;
    L_Last_First_Fault_Source : INT;
    L_Last_Root_Cause : E_System_Root_Cause;
    L_History_Event : ST_History_Record;
    L_History_Write_Event : BOOL;
    L_Last_Operator_Journal_Seq : UDINT;
    L_Last_Event_Code : UDINT;
    L_Last_Event_Value : REAL;
    L_Last_Event_Time_MS : UDINT;
    L_Gateway_Writes_Allowed : BOOL;

    L_Scenario_Req_Operator : E_SCENARIO_TYPE;
    L_Scenario_Req_Gateway  : E_SCENARIO_TYPE;
    L_Scenario_Req_Rule     : E_SCENARIO_TYPE;
    L_Scenario_Req_Final    : E_SCENARIO_TYPE; // TRACE ONLY: arbitration result before policy
    L_Scenario_Intent       : E_SCENARIO_TYPE;
L_Scenario_Source       : E_SCENARIO_SOURCE;
L_Scenario_Changed      : BOOL;
L_Last_Scenario_Change_Time : UDINT;

L_IO_Fault_Prev : BOOL;
L_Comm_Fault_Prev : BOOL;
L_Sensor_Fault_Prev : BOOL;
L_Subsystem_Fault_Prev : BOOL;
L_Mode_Prev : E_System_Operating_Mode;
L_User_Access_Denied_Prev : BOOL;

    L_Persist_Buffer : ARRAY[0..4] OF BYTE;
    L_Last_Written_Persist_Buffer : ARRAY[0..4] OF BYTE;
    L_Persist_Buffer_Changed : BOOL;
    L_Last_Persist_Write_MS : UDINT;
    L_Recovery_Done : BOOL;
    L_Persist_Struct : ST_Persist;
END_VAR

// ... (content unchanged until target section)

// === STAGE I2b: FINAL USER INTENT PUBLICATION ===
GVL_INTENT_USER.I_Scenario_Request := L_Scenario_Req_Gateway;
GVL_INTENT_USER.I_Dangerous_Action_Request := GVL_COMMAND.CMD_Dangerous_Action_Request;
GVL_INTENT_USER.I_Dangerous_Action_Confirm := GVL_COMMAND.CMD_Dangerous_Action_Confirm;
GVL_INTENT_USER.I_User_Access_Level := GVL_COMMAND.CMD_User_Access_Level;
GVL_INTENT_USER.I_Water_Valve_Test_Open := GVL_COMMAND.CMD_Water_Valve_Test_Open;
GVL_INTENT_USER.I_Water_Valve_Test_Close := GVL_COMMAND.CMD_Water_Valve_Test_Close;
GVL_INTENT_USER.I_Water_Valve_Test_Confirm := GVL_COMMAND.CMD_Water_Valve_Test_Confirm;
GVL_INTENT_USER.I_Gas_Valve_Test_Open := GVL_COMMAND.CMD_Gas_Valve_Test_Open;
GVL_INTENT_USER.I_Gas_Valve_Test_Close := GVL_COMMAND.CMD_Gas_Valve_Test_Close;
GVL_INTENT_USER.I_Gas_Valve_Test_Confirm := GVL_COMMAND.CMD_Gas_Valve_Test_Confirm;
GVL_INTENT_USER.I_Water_Selective_Recover := GVL_COMMAND.CMD_Water_Selective_Recover;
GVL_INTENT_USER.I_Gas_Selective_Recover := GVL_COMMAND.CMD_Gas_Selective_Recover;

// >>> BULK_SYNC_ANCHOR: PRG_System <<<
